TYPE ST_SEW_MoviC_Velocity_Config :
STRUCT
	bForceMode				: BOOL; //Ignore process data from fieldbus.
	bSwapProcessData		: BOOL; //Reverse process data byte order from/to fieldbus.
	nSoftwareLimitMin		: DINT := -2147483648;	//Position limit minimum in LU
	nSoftwareLimitMax		: DINT := 2147483647;	//Position limit maximum in LU
	nReferencePos			: DINT := 0;			//Reference position in LU when using mode 300
	fDecCoastStop			: REAL := 1000.0;		//Deceleration for coast/brake stop in LU/s^2
	fDecEstop				: REAL := 100.0;		//Deceleration for emergency stop in LU/s^2
	fDecelerationLimit		: REAL := 100.0;		//Decceleration limit (bus stop) in LU/s^2
	fRatioVelocity			: REAL := 1.0;			//Ratio for setpoint velocity
	fRatioAccDec			: REAL := 1.0;			//Ratio for setpoint acceleration/deceleration
	fRatioPosition			: REAL := 1.0;			//Ratio for position output
	nJerk					: INT  := 0;			//Jerk from 0 to 100%
	fPositionOffset			: REAL := 0;
	fInitPosition			: REAL := 0;
	fResolution				: REAL := 0.1;
	bOutputVelocity			: BOOL := TRUE;			//TRUE: TargetValue = Velocity, FALSE: TargetValue = Position
END_STRUCT
END_TYPE

(* stored: Version 1.1.0.1, ProductVersion 3.1.4024.12
   DUT ST_SEW_MoviC_Velocity_Config: Id {97c4e567-bbd9-0c89-2d14-841138991a08} *)
